(* CoDeSys 2.3 export: GLOBAL_VARIABLES.EXP *)

(* Global variable list: Global_Variables *)
VAR_GLOBAL
	xActuatorReady		: BOOL;	(* In Position *)
	wActuatorStatus		: WORD;	(* Current Status *)
	wActuatorPosition	: WORD;	(* Current Position *)
	wActuatorAlarm		: WORD;	(* Current Alarm *)
END_VAR
VAR_GLOBAL RETAIN
	wActuatorTarget		: WORD;	(* Target Position *)
END_VAR
